(* CoDeSys 2.3.9.50 project: CFA4.pro *)
(* Libraries: STANDARD.LIB 5.6.98 11:03:02 *)

(* Task configuration *)
TASK Standard (PRIORITY := 0, INTERVAL := T#10ms);
	MAIN
END_TASK

(* Global variable list: Global_Variables *)
VAR_GLOBAL
(* Machine Condition *)
	MC							:ST_MC;
(* ST10 I/O*)
	I10_Housing_Present		AT%I*	 : BOOL;
	I10_Cover_Present		AT%I*	 : BOOL;
	I10_Curtain_Safety 		AT%I*	 :BOOL;

(* Error *)
	E10_ProductPresent		 : BOOL;


(* XTS Variable*)
	CarStation 					: ARRAY[0..20] OF ST_Car;
	T10_Bypass					: BOOL;
	T20_Bypass: BOOL;
END_VAR

(* Data type *)
TYPE ST_Car :
STRUCT
	WP_Num_ID:DINT;
	WP_Present:BOOL; (*P1 Part Memory*)
	WP_Status:BOOL;	(*Overall Status Pass*)
	Result : ARRAY[0..200] OF BOOL;
	Done : ARRAY[0..200]OF BOOL;
	Press_Final_Force:REAL;
	Press_Final_Pos:REAL;
END_STRUCT
END_TYPE

(* Data type *)
TYPE ST_MC :
STRUCT
	Autorun					: BOOL;
	DryRun					: BOOL;
	ManualMode				: BOOL;
END_STRUCT
END_TYPE

(* Data type *)
TYPE ST_Station :
STRUCT
	Autorun_Cond		: BOOL;
	NextStep				: BOOL;
	Autorun				: BOOL;
	Done				: BOOL;
	SingleStep			: BOOL;
	SingleStepMode		: BOOL;
	OneCycleMode		: BOOL;
	OneCycle			: BOOL;
	Origin				: BOOL;
	inPosition			: BOOL;
	Bypass				: BOOL;
	Car					: INT;

	E_MinorError			: BOOL;
	E_MajorError			: BOOL;



END_STRUCT
END_TYPE

(* POU MAIN, ST *)
PROGRAM MAIN
VAR
END_VAR
(*ST10*)
ST10_Main;

(*ST20*)
ST20_Main;
END_PROGRAM

(* POU ST10_Main, ST *)
PROGRAM ST10_Main
VAR

(*ST10 condition*)
	ST10					: ST_Station;
	S10_CurtainClear			: BOOL;
	F10_ClearDone_Trig		: R_TRIG;
	F10_CurtainClear_Trig		: R_TRIG;

(*Local Status*)
	curr_state				: INT;
	next_state				: INT;
	X						: INT;

END_VAR
(************************************************************************************************************************************
*
*										station control 
*
************************************************************************************************************************************)

ST10.Autorun 			:= 	MC.Autorun OR MC.DryRun OR ST10.SingleStepMode OR ST10.OneCycleMode;
ST10.Autorun_Cond	:= 	NOT ST10.Done AND ST10.inPosition AND NOT MC.ManualMode;
ST10.NextStep		:= 	ST10.Autorun OR MC.DryRun OR ST10.SingleStep OR ST10.OneCycle;
ST10.Origin			:=	ST10.inPosition;
ST10.Bypass			:=	T10_Bypass;

(************************************************************************************************************************************
*
*								clear done when new car arrive
*
************************************************************************************************************************************)
F10_ClearDone_Trig(CLK:=ST10.inPosition , Q=> );
IF F10_ClearDone_Trig.Q THEN
	ST10.Done 						:= FALSE;
END_IF


(************************************************************************************************************************************
*
*										reset all done
*
***********************************************************************************************************************************)

IF F10_ClearDone_Trig.Q THEN
	FOR X:=1 TO 200 BY 10 DO
		CarStation[ST10.Car].Done[x]	:= FALSE;
		CarStation[ST10.Car].Result[x] 	:= FALSE;
	END_FOR
END_IF


(************************************************************************************************************************************
*
*										Curtain Clear
*
************************************************************************************************************************************)
F10_CurtainClear_Trig(CLK:=I10_Curtain_Safety , Q=> );
S10_CurtainClear := F10_CurtainClear_Trig.Q;



(************************************************************************************************************************************
*
*										Station Action
*
************************************************************************************************************************************)
Auto;
Error;
Origin;
END_PROGRAM
ACTION Auto:
(************************************************************************************************************************************
*
* 								add ST10_done Result
*
************************************************************************************************************************************)
IF ST10.Done THEN
	CarStation[ST10.Car].Done[10]		:= TRUE;
	CarStation[ST10.Car].Result[10]		:= TRUE;
END_IF


(************************************************************************************************************************************
*
*						case only run after sufficient condition stated here
*
************************************************************************************************************************************)
IF ST10.NextStep AND ST10.Autorun_Cond AND ST10.Autorun  THEN
	curr_state := next_state;
	ST10.SingleStep := FALSE;
ELSE
	curr_state := 0;
END_IF


(************************************************************************************************************************************
*
*											CASE
*
************************************************************************************************************************************)

CASE curr_state OF
0:
 (*check for present cover, here dont need starting condition because the curr_state condition already guard it*)
	IF I10_Housing_Present OR I10_Cover_Present THEN
		E10_ProductPresent := TRUE;
	ELSE
		next_state := next_state + 10;
	END_IF
10:
(*wait for product load*)
	IF S10_CurtainClear AND ((I10_Housing_Present AND I10_Cover_Present) OR MC.DryRun) THEN
		next_state := 0;
		ST10.Done := TRUE;
		ST10.OneCycle := FALSE;
	END_IF
END_CASE
END_ACTION
ACTION Error:
(************************************************************************************************************************************
*
*										station error  
*
************************************************************************************************************************************)
ST10.E_MinorError := E10_ProductPresent;
END_ACTION
ACTION Origin:
(***********************************************************************************************************************************
*
*										station origin 
*
************************************************************************************************************************************)
(*there is no action for origin for station 1*)
ST10.Origin 			:= ST10.inPosition;
END_ACTION

(* POU ST20_Main, ST *)
PROGRAM ST20_Main
VAR

(*ST10 condition*)
	ST20					: ST_Station;
	S20_CurtainClear			: BOOL;
	F20_ClearDone_Trig		: R_TRIG;
	F20_CurtainClear_Trig		: R_TRIG;

(*Local Status*)
	curr_state				: INT;
	next_state				: INT;
	X						: INT;

END_VAR
(************************************************************************************************************************************
*
*										station control 
*
************************************************************************************************************************************)

ST20.Autorun 			:= 	MC.Autorun OR MC.DryRun OR ST20.SingleStepMode OR ST20.OneCycleMode;
ST20.Autorun_Cond	:= 	NOT ST20.Done AND ST20.inPosition AND NOT MC.ManualMode;
ST20.NextStep		:= 	ST20.Autorun OR MC.DryRun OR ST20.SingleStep OR ST20.OneCycle;
ST20.Origin			:=	ST20.inPosition;
ST20.Bypass			:=	T20_Bypass;

(************************************************************************************************************************************
*
*								clear done when new car arrive
*
************************************************************************************************************************************)
F20_ClearDone_Trig(CLK:=ST20.inPosition , Q=> );
IF F20_ClearDone_Trig.Q THEN
	ST20.Done 						:= FALSE;
END_IF


(************************************************************************************************************************************
*
*										reset all done
*
***********************************************************************************************************************************)

IF F20_ClearDone_Trig.Q THEN
	FOR X:=1 TO 200 BY 10 DO
		CarStation[ST20.Car].Done[x]	:= FALSE;
		CarStation[ST20.Car].Result[x] 	:= FALSE;
	END_FOR
END_IF


(************************************************************************************************************************************
*
*										Curtain Clear
*
************************************************************************************************************************************)
F20_CurtainClear_Trig(CLK:=I10_Curtain_Safety , Q=> );
S20_CurtainClear := F20_CurtainClear_Trig.Q;



(************************************************************************************************************************************
*
*										Station Action
*
************************************************************************************************************************************)
Auto;
Error;
Origin;
END_PROGRAM
ACTION Auto:
(************************************************************************************************************************************
*
* 								add ST20_done Result
*
************************************************************************************************************************************)
IF ST20.Done THEN
	CarStation[ST20.Car].Done[10]		:= TRUE;
	CarStation[ST20.Car].Result[10]		:= TRUE;
END_IF


(************************************************************************************************************************************
*
*						case only run after sufficient condition stated here
*
************************************************************************************************************************************)
IF ST20.NextStep AND ST20.Autorun_Cond AND ST20.Autorun  THEN
	curr_state := next_state;
	ST20.SingleStep := FALSE;
ELSE
	curr_state := 0;
END_IF


(************************************************************************************************************************************
*
*											CASE
*
************************************************************************************************************************************)

CASE curr_state OF
0:
 (*check for present cover, here dont need starting condition because the curr_state condition already guard it*)
	IF I10_Housing_Present OR I10_Cover_Present THEN
		E10_ProductPresent := TRUE;
	ELSE
		next_state := next_state + 10;
	END_IF
10:
(*wait for product load*)
	IF S20_CurtainClear AND ((I10_Housing_Present AND I10_Cover_Present) OR MC.DryRun) THEN
		next_state := 0;
		ST20.Done := TRUE;
		ST20.OneCycle := FALSE;
	END_IF
END_CASE
END_ACTION
ACTION Error:
(************************************************************************************************************************************
*
*										station error  
*
************************************************************************************************************************************)
ST20.E_MinorError := E10_ProductPresent;
END_ACTION
ACTION Origin:
(***********************************************************************************************************************************
*
*										station origin 
*
************************************************************************************************************************************)
(*there is no action for origin for station 1*)
ST20.Origin 			:= ST20.inPosition;
END_ACTION
